// TIA Portal V20 export
DATA_BLOCK "LBP_Internal3"   // DB25002
TITLE = Internal DB for basic program / DB interne pour programme de base
// DB only for internal use in the basic program / DB réservé à l'utilisation interne dans le programme de base
// stored: InstanceOfName LBP_InternalProc8, InstanceOfType FB
"LBP_InternalProc8"
   // VAR
   //    statPlcCtrlsNm1 { ExternalAccessible := 'False'; ExternalVisible := 'False'; ExternalWritable := 'False'} : Bool;
   //    statDateAndTime { ExternalAccessible := 'False'; ExternalVisible := 'False'; ExternalWritable := 'False'} : Date_And_Time;
   //    statLastSecond { ExternalAccessible := 'False'; ExternalVisible := 'False'; ExternalWritable := 'False'} : Byte;
   // END_VAR
BEGIN
END_DATA_BLOCK
